// TIA Portal V17 export
// export: Created 2025-06-25T13:13:01.8055431Z, ExportSetting WithDefaults, DisplayName Totally Integrated Automation Portal, DisplayVersion V17 Update 8, DisplayName TIA Portal Openness, DisplayVersion V17 Update 8, DisplayName TIA Portal Version Control Interface, DisplayVersion V17, DisplayName STEP 7 Professional, DisplayVersion V17 Update 8, DisplayName STEP 7 Safety, DisplayVersion V17 Update 6, DisplayName WinCC Advanced, DisplayVersion V17 Update 8
ORGANIZATION_BLOCK "Main"   // OB1, FBD, ProgramCycle
TITLE = "Main Program Sweep (Cycle)"
{ S7_Optimized_Access := 'TRUE' }
VERSION : 0.1
// stored: AutoNumber true, IsIECCheckEnabled false, SetENOAutomatically false
   VAR_INPUT
      Initial_Call : Bool;   // Initial call of this OB
      Remanence : Bool;   // =True, if remanent data are available
   END_VAR
   VAR_TEMP
      dummy : Bool;
      InitError : Bool;
      RetVal10 : LReal;
   END_VAR
BEGIN

REGION Network 1: First cycle. Used for initialization
   // Use SET so that .bFirstCycle can be manually triggered
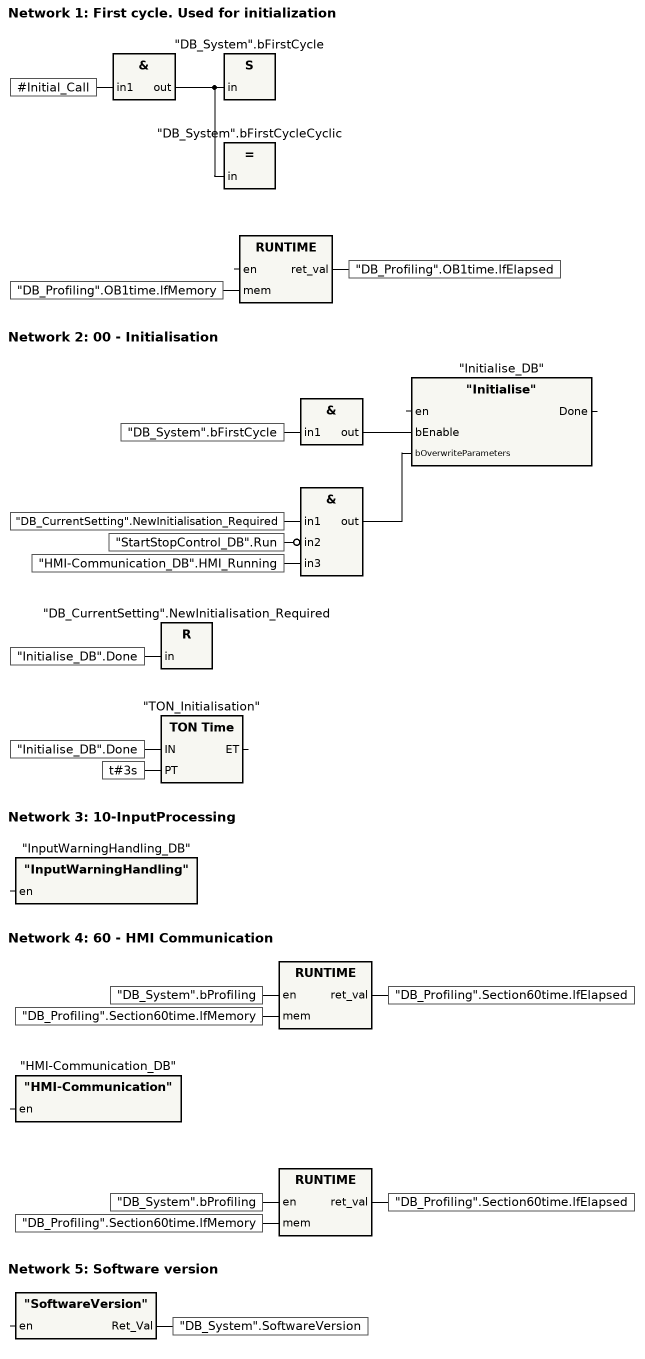
   // no SCL statement known for Runtime: written as a call
   IF #Initial_Call THEN "DB_System".bFirstCycle := TRUE; END_IF;
   "DB_System".bFirstCycleCyclic := #Initial_Call;
   "DB_Profiling".OB1time.lfElapsed := Runtime(mem := "DB_Profiling".OB1time.lfMemory);
END_REGION

REGION Network 2: 00 - Initialisation
   // Update alarm limits from DB_CurrentSettings on every restart
   // Load a new DB_CurrentSetting on NewInitialisation_Required, and update the alarm limits
   "Initialise_DB"(bEnable := "DB_System".bFirstCycle,   // "Initialise"
                   bOverwriteParameters := "DB_CurrentSetting".NewInitialisation_Required AND NOT "StartStopControl_DB".Run AND "HMI-Communication_DB".HMI_Running);
   IF "Initialise_DB".Done THEN "DB_CurrentSetting".NewInitialisation_Required := FALSE; END_IF;
   "TON_Initialisation".TON(IN := "Initialise_DB".Done, PT := t#3s);
END_REGION

REGION Network 3: 10-InputProcessing
   "InputWarningHandling_DB"();   // "InputWarningHandling"
END_REGION

REGION Network 4: 60 - HMI Communication
   // no SCL statement known for Runtime: written as a call
   IF "DB_System".bProfiling THEN
       "DB_Profiling".Section60time.lfElapsed := Runtime(mem := "DB_Profiling".Section60time.lfMemory);
   END_IF;
   "HMI-Communication_DB"();   // "HMI-Communication"
   IF "DB_System".bProfiling THEN
       "DB_Profiling".Section60time.lfElapsed := Runtime(mem := "DB_Profiling".Section60time.lfMemory);
   END_IF;
END_REGION

REGION Network 5: Software version
   "DB_System".SoftwareVersion := "SoftwareVersion"();
END_REGION

REGION Network 6: Reset first cycle
   // This network must be the last one in the program
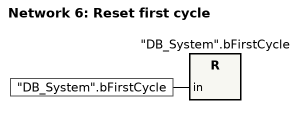
   IF "DB_System".bFirstCycle THEN "DB_System".bFirstCycle := FALSE; END_IF;
END_REGION
END_ORGANIZATION_BLOCK
